FUNCTION_BLOCK FB_LiftA EXTENDS FB_Lift
VAR_INPUT
END_VAR
VAR_OUTPUT
END_VAR
VAR
END_VAR

END_FUNCTION_BLOCK

(* stored: Version 1.1.0.1
   POU FB_LiftA: Id {5c11f934-409c-4a47-af7d-811380022bc6}, SpecialFunc None *)
